{attribute 'qualified_only'}
{attribute 'strict'}
TYPE  E_SensorStatus :
(
	SENSOR_OK       := 0,
    SENSOR_WARNING  := 1,
    SENSOR_ALARM    := 2,
    SENSOR_FAULT    := 3,
    SENSOR_BYPASS   := 4
);
END_TYPE

(* stored: Version 1.1.0.1, ProductVersion 3.1.4024.16
   DUT E_SensorStatus: Id {4f80d977-33be-48a2-9976-ef730d6f4d0b} *)
